120: // If counter is equal to the max # of test channels, reset it; else, proceed around again 
IF (uiLoopRcvIndex = gc.uiMaxNrDMXTestCh) THEN
	iCompareSeq[ENUM_SeqSM.Once]			:= 130;
ELSE
	uiLoopRcvIndex							:= uiLoopRcvIndex +1;
	//Next iteration
	tonTestIterGap.IN						:= TRUE;
	iCompareSeq[ENUM_SeqSM.Once]			:= 10;
 (*iCounter <> gc.usiMaxNrOfChannels*)
END_IF

130:
xDMXSeqTestInProgressOnce					:= FALSE;
iCompareSeq[ENUM_SeqSM.Once]				:= 140;

140:
IF rt_ResetTestSeq.Q AND NOT rt_RunSeqTestOnce.Q THEN
	FOR uiCounter2 := 0 TO gc.uiMaxNrDMXTestCh BY 1 DO 
		arr_diTestPNPSeqOnceLine[uiCounter2]		:= 0;
		arr_diTestNPNSeqOnceLine[uiCounter2]		:= 0;
//		arrdiTestPNPSeqOnceComplete[uiCounter2]		:= 0;
//		arrdiTestNPNSeqOnceComplete[uiCounter2]		:= 0;
		arrdiTestNPNSeqOnceCompleteProblemIndex[uiCounter2]	:= 0;
	END_FOR
	diCompTestResult							:= 0;
	iCompareSeq[ENUM_SeqSM.Once]				:= 0; (* reset to beginning *)
END_IF

END_CASE
END_ACTION

ACTION SeqTestOnceDC:
//Run Once - DMX Channels only for now

rt_RunSeqTestOnceDC();
rt_ResetTestSeqDC();

CASE iCompareSeq[ENUM_SeqSM.OnceDC] OF
	
0: // If test is triggered by user
//Trigger should be something like 
IF rt_RunSeqTestOnceDC.Q THEN
	xDMXSeqTestInProgressOnceDC				:= TRUE;
	uiLoopRcvIndex							:= cuiMinDUTIndex; 
	iCompareSeq[ENUM_SeqSM.OnceDC]			:= 10;
END_IF

10: // Zero out all comparison buffers before each comparison
IF (uiLoopRcvIndex=0) THEN
	IF xDMXSeqTestInProgressOnceDC THEN
//by default, Counter = 0 at the first initialization; it is reset at the end of this State Machine
//Clear Storage Buffers pre-test to ensure no old data interferes with current test
		FOR uiCounter4 := 0 TO gc.uiMaxNrDMXTestCh BY 1 DO
			arrxExpctdTmpPNPSeqDC[uiCounter4]		:= 0;		//should be all 0s ; PNP<>DMX
			arrxExpctdTmpNPNSeqDC[uiCounter4]		:= 0;
//			arrxExpctdTmpPNPSeqDC[uiCounter4]		:= 0;		
//			arrxExpctdTmpNPNSeqDC[uiCounter4]		:= 0;
			arrxRcvdBufferPNPSeq[uiCounter4]		:= 0;		//should be all 0s too ; PNP<>DMX	
			arrxRcvdBufferNPNSeq[uiCounter4]		:= 0;			
			g_ast.DMX[uiCounter4].IQ.xCmdOff		:= TRUE;	
		END_FOR
	iCompareSeq[ENUM_SeqSM.OnceDC]					:= 20;
	END_IF
ELSIF (uiLoopRcvIndex>0) THEN // to avoid 
	IF xDMXSeqTestInProgressOnceDC AND tonTestIterGap.Q THEN
		tonTestIterGap.IN	:= FALSE;
		//by default, Counter = 0 at the first initialization; it is reset at the end of this State Machine
		//Clear Storage Buffers pre-test to ensure no old data interferes with current test
		FOR uiCounter4 := 0 TO gc.uiMaxNrDMXTestCh BY 1 DO
			arrxExpctdTmpPNPSeqDC[uiCounter4]		:= 0;		//should be all 0s - PNP<>DMX
			arrxExpctdTmpNPNSeqDC[uiCounter4]		:= 0;
			arrxRcvdBufferPNPSeq[uiCounter4]		:= 0;		
			arrxRcvdBufferNPNSeq[uiCounter4]		:= 0;		
		END_FOR
		
	iCompareSeq[ENUM_SeqSM.OnceDC]					:= 25; // don't write the hardware value (skip 20)
	END_IF	
END_IF
	
20:	
//write 'hardware-clear' state 
g_ast.DMXHWOut									:= g_ast.DMXPhysOut;

iCompareSeq[ENUM_SeqSM.OnceDC]					:= 25;

25:
//Copy static test indices from Expected_Static - as these should still be used for comparisons
//FOR uiCounter4 := 0 TO gc.uiMaxNrDMXTestCh BY 1 DO
//	IF (arrui24VTestIndices[uiCounter4] <> 0) THEN	
		MEMCPY(srcAddr:=ADR(arrxExpctdTmpPNP24V[cuiMinDUTIndex]),destAddr:=ADR(arrxExpctdTmpPNPSeqDC[cuiMinDUTIndex]),n:=gc.uiChannelsUT);
//		MEMCPY(srcAddr:=ADR(arrxExpctdTmpNPN24V[cuiMinDUTIndex]),destAddr:=ADR(arrxExpctdTmpNPNSeqDMX[cuiMinDUTIndex]),n:=gc.uiChannelsUT);
//		MEMCPY(srcAddr:=ADR(arrxExpctdTmpPNP24V[arrui24VTestIndices[uiCounter4]]),destAddr:=ADR(arrxExpctdTmpPNPSeqDC[arrui24VTestIndices[uiCounter4]]),n:=1);
//		MEMCPY(srcAddr:=ADR(arrxExpctdTmpNPN24V[arrui24VTestIndices[uiCounter4]]),destAddr:=ADR(arrxExpctdTmpNPNSeqDC[arrui24VTestIndices[uiCounter4]]),n:=1);
//	END_IF
	
//	IF (arruiGNDTestIndices[uiCounter4] <> 0) THEN	
//		MEMCPY(srcAddr:=ADR(arrxExpctdTmpPNPGND[cuiMinDUTIndex]),destAddr:=ADR(arrxExpctdTmpPNPSeqDMX[cuiMinDUTIndex]),n:=gc.uiChannelsUT);
		MEMCPY(srcAddr:=ADR(arrxExpctdTmpNPNGND[cuiMinDUTIndex]),destAddr:=ADR(arrxExpctdTmpNPNSeqDC[cuiMinDUTIndex]),n:=gc.uiChannelsUT);
//		MEMCPY(srcAddr:=ADR(arrxExpctdTmpPNPGND[arruiGNDTestIndices[uiCounter4]]),destAddr:=ADR([arrxExpctdTmpPNPSeqDC[uiCounter4]]),n:=1);
//		MEMCPY(srcAddr:=ADR(arrxExpctdTmpNPNGND[arruiGNDTestIndices[uiCounter4]]),destAddr:=ADR(arrxExpctdTmpNPNSeqDC[arruiGNDTestIndices[uiCounter4]]),n:=1);
//	END_IF
//END_FOR

// Be careful not to overstamp existing arrays!  Right now MEMCPY is only addressing PNP24V & NPNGND

iCompareSeq[ENUM_SeqSM.OnceDC]					:= 30;

30: //Set the Expected Mask & write data to controller
//Write the first index from the specified array of indices
IF (arruiSeqTestIndicesDC[uiLoopRcvIndex] <> 0) THEN
//Also copy this specific channel index value to the comparison array
	
//Don't copy NPN indices for DC; this doesn't generally make sense
	MEMCPY(srcAddr:=ADR(arrxExpctdTmpPNP[arruiSeqTestIndicesDC[uiLoopRcvIndex]]),destAddr:=ADR(arrxExpctdTmpPNPSeqDC[arruiSeqTestIndicesDC[uiLoopRcvIndex]]),n:=SIZEOF(arrxExpctdTmpPNP[arruiSeqTestIndicesDC[uiLoopRcvIndex]]));
//	MEMCPY(srcAddr:=ADR(arrxExpctdTmpNPN[arruiSeqTestIndicesDMX[uiLoopRcvIndex]]),destAddr:=ADR(arrxExpctdTmpNPNSeqDMX[arruiSeqTestIndicesDMX[uiLoopRcvIndex]]),n:=SIZEOF(arrxExpctdTmpNPN[arruiSeqTestIndicesDMX[uiLoopRcvIndex]]));	
	
	//And Cmd - turn on - that respective channel
	g_ast.DMX[arruiSeqTestIndicesDC[uiLoopRcvIndex]].IQ.xCmdOn			:= TRUE;
	FOR uiCounter3 := cuiMinDUTIndex TO gc.uiMaxNrDMXTestCh BY 1 DO
		IF uiCounter3 <> arruiSeqTestIndicesDC[uiLoopRcvIndex] THEN
			g_ast.DMX[uiCounter3].IQ.xCmdOff	:= TRUE;	
		END_IF
	END_FOR
ELSIF (arruiSeqTestIndicesDC[uiLoopRcvIndex] = 0) THEN
	FOR uiCounter3 := cuiMinDUTIndex TO gc.uiMaxNrDMXTestCh BY 1 DO
		IF uiCounter3 <> arruiSeqTestIndicesDC[uiLoopRcvIndex] THEN
			g_ast.DMX[uiCounter3].IQ.xCmdOff	:= TRUE;	
		END_IF
	END_FOR
END_IF

iCompareSeq[ENUM_SeqSM.OnceDC]		:= 35;

35:
//Write to hardware
g_ast.DMXHWOut						:= g_ast.DMXPhysOut;

iCompareSeq[ENUM_SeqSM.OnceDC]		:= 40;

40:
//Write DMX channels
tonWriteCopyWait.IN					:= TRUE;
iCompareSeq[ENUM_SeqSM.OnceDC]		:= 50;

50:
IF tonWriteCopyWait.Q THEN
	tonWriteCopyWait.IN				:= FALSE;
	iCompareSeq[ENUM_SeqSM.OnceDC]	:= 60;
END_IF

60:
//IF there is an index for a 'Light' element, then copy that element's value to a new pair of arrays, for 'Received'
//IF arruiSeqTestIndicesDMX[uiLoopRcvIndex] <> 0 THEN
(*
FOR uiCounter6 := 0 TO gc.uiMaxNrDMXTestCh BY 1 DO 
	arr_udiMEMCPYPNPSeqOnceRcvdTmp[uiCounter6]	:= MEMCPY(srcAddr:=ADR(arrxTestChInputPNPAlias[uiCounter6]),destAddr:=ADR(arrxRcvdBufferPNPSeq[uiCounter6]),n:=SIZEOF(arrxTestChInputPNP[uiCounter6])); //bytes
	arr_udiMEMCPYNPNSeqOnceRcvdTmp[uiCounter6]	:= MEMCPY(srcAddr:=ADR(arrxTestChInputNPNAlias[uiCounter6]),destAddr:=ADR(arrxRcvdBufferNPNSeq[uiCounter6]),n:=SIZEOF(arrxTestChInputNPN[uiCounter6])); //bytes)
	//	MEMCPY(srcAddr:=ADR(arrxExpctdTmpPNP[arruiSeqTestIndices[uiLoopRcvIndex]]),destAddr:=ADR(arrxExpctdTmpPNPSeq[arruiSeqTestIndices[uiLoopRcvIndex]]),n:=1); //bytes
	//	MEMCPY(srcAddr:=ADR(arrxExpctdTmpNPN[arruiSeqTestIndices[uiLoopRcvIndex]]),destAddr:=ADR(arrxExpctdTmpNPNSeq[arruiSeqTestIndices[uiLoopRcvIndex]]),n:=1); //bytes
END_FOR
*)
//Stash
//arr_udiMEMCPYPNPSeqOnceRcvd	:= arr_udiMEMCPYPNPSeqOnceRcvdTmp;
//arr_udiMEMCPYNPNSeqOnceRcvd	:= arr_udiMEMCPYNPNSeqOnceRcvdTmp;

//END_IF

//We should also 'expect' the static indices - and if we passed the static test already - they will still be on, so grab and add those to the 'Expected' Buffer
//This is a gate to leave this state; the MEMCPY operation had to return for all values
	
(*
70:
tonReadWait.IN							:= TRUE;
iCompareSeq[ENUM_SeqSM.OnceDC]			:= 80;

80: // if wait completed, set the bit for conversion high
//Conversion Function call
IF tonReadWait.Q THEN
	tonReadWait.IN					:= FALSE;
	iCompareSeq[ENUM_SeqSM.OnceDC]	:= 90;
END_IF
*)

90:
//Run Comparos
IF iCompareStaticSM <> 90 THEN //because it uses the same iterator in StaticSM - shouldn't be the case, but this is a safeguard
	FOR uiCounter6	:= 0 TO gc.uiMaxNrDMXTestCh BY 1 DO
		arr_diTestPNPSeqOnceLineTmp[uiCounter6]			:= MEMCMP(pBuf1:=ADR(arrxExpctdTmpPNPSeqDC[uiCounter6]),pBuf2:=ADR(arrxRcvdBufferPNPSeq[uiCounter6]),n:=SIZEOF(arrxExpctdTmpPNPSeqDC[uiCounter6]));
//		arr_diTestNPNSeqOnceLineTmp[uiCounter6]			:= MEMCMP(pBuf1:=ADR(arrxExpctdTmpNPNSeqDMX[uiCounter6]),pBuf2:=ADR(arrxRcvdBufferNPNSeq[uiCounter6]),n:=SIZEOF(arrxExpctdTmpNPNSeqDMX[uiCounter6])); 
		arrdiTestPNPSeqOnceCompleteTmp[uiCounter6]		:= MEMCMP(pBuf1:=ADR(arrxExpctdTmpPNPSeqDC[cuiMinDUTIndex]),pBuf2:=ADR(arrxRcvdBufferPNPSeq[cuiMinDUTIndex]),n:=gc.uiChannelsUT); //UINTs are 16-bit/2 bytes
//		arrdiTestNPNSeqOnceCompleteTmp[uiCounter6]		:= MEMCMP(pBuf1:=ADR(arrxExpctdTmpNPNSeqDMX[cuiMinDUTIndex]),pBuf2:=ADR(arrxRcvdBufferNPNSeq[cuiMinDUTIndex]),n:=gc.uiChannelsUT); //UINTs are 16-bit/2 bytes
	END_FOR
arr_diTestPNPSeqOnceLine	:= arr_diTestPNPSeqOnceLineTmp;
arrdiTestPNPSeqOnceComplete	:= arrdiTestPNPSeqOnceCompleteTmp;
	
END_IF

(* log the error index 
IF arr_diTestPNPSeqOnce[uiLoopRcvIndex] <> 0 THEN
	memcpy(srcAddr:=uiLoopRcvIndex,destAddr:=, n:=2)
END_IF
*)

iCompareSeq[ENUM_SeqSM.OnceDC]				:= 100;

100: // If counter is equal to the max # of test channels, reset it; turn off the DMX channels that were turned on in the course of the test

IF (uiLoopRcvIndex = gc.uiMaxNrDMXTestCh) THEN
	iCompareSeq[ENUM_SeqSM.OnceDC]			:= 110;
ELSE
	uiLoopRcvIndex							:= uiLoopRcvIndex +1;
	//Next iteration
	tonTestIterGap.IN						:= TRUE;
	iCompareSeq[ENUM_SeqSM.OnceDC]			:= 10;
 (*iCounter <> gc.usiMaxNrOfChannels*)
END_IF

110:
xDMXSeqTestInProgressOnceDC					:= FALSE;
iCompareSeq[ENUM_SeqSM.OnceDC]				:= 120;

120:
IF rt_ResetTestSeqDC.Q AND NOT rt_RunSeqTestOnceDC.Q THEN
	FOR uiCounter2 := 0 TO gc.uiMaxNrDMXTestCh BY 1 DO 
		arr_diTestPNPSeqOnceLine[uiCounter2]		:= 0;
		arr_diTestNPNSeqOnceLine[uiCounter2]		:= 0;
		arrdiTestPNPSeqOnceComplete[uiCounter2]		:= 0;
		arrdiTestNPNSeqOnceComplete[uiCounter2]		:= 0;
	END_FOR
	diCompTestResult							:= 0;
	iCompareSeq[ENUM_SeqSM.OnceDC]				:= 0; (* reset to beginning *)
END_IF

END_CASE
END_ACTION

END_PROGRAM

// ---- POUs/FunctionBlocks/HelperPRG/InterfaceLink.TcPOU
PROGRAM InterfaceLink
VAR
	iResult					: INT;
	iLoopFBAnalogIn			: INT;
	iLoopFBSensor			: INT;
	iLoopFBValveSensor		: INT;
	iLoopFBDigCtrl			: INT;
	iLoopFBValveCtrl		: INT;
	uiLoopDMXCtrlI			: UINT;
	uiLoopDMXCtrlII			: UINT;
	uiLoopDebouncePNPI		: UINT;
	uiLoopDebounceNPNI		: UINT;
END_VAR

//Call all the I/O Function Blocks continuously; link to array-structs with every call;
(*
FOR iLoopFBAnalogIn := 0 TO gc.usiMaxNrOfAnalogIn BY 1 DO
	gFB.arrFB_AnalogInput[iLoopFBAnalogIn](I:=gast_AnalogInput[iLoopFBAnalogIn].I, IQ:=gast_AnalogInput[iLoopFBAnalogIn].IQ, Q=>gast_AnalogInput[iLoopFBAnalogIn].Q);
END_FOR

FOR iLoopFBSensor := 0 TO gc.usiMaxNrOfSensor BY 1 DO
	gFB.arrFB_Sensor[iLoopFBSensor](I:=gast_SensorInput[iLoopFBSensor].I, IQ:=gast_SensorInput[iLoopFBSensor].IQ, Q=>gast_SensorInput[iLoopFBSensor].Q);
END_FOR

FOR iLoopFBValveSensor := 0 TO (2*gc.usiMaxNrOfValveCtrl) BY 1 DO
	gFB.arrFB_Sensor[iLoopFBValveSensor](I:=gast_ValveSensorInput[iLoopFBValveSensor].I, IQ:=gast_ValveSensorInput[iLoopFBValveSensor].IQ, Q=>gast_ValveSensorInput[iLoopFBValveSensor].Q);
END_FOR

FOR iLoopFBDigCtrl := 0 TO gc.usiMaxNrOfSensor BY 1 DO
	gFB.arrFB_DigCtrl[iLoopFBDigCtrl](I:=gast_DigCtrlOutput[iLoopFBDigCtrl].I, IQ:=gast_DigCtrlOutput[iLoopFBDigCtrl].IQ, Q=>gast_DigCtrlOutput[iLoopFBDigCtrl].Q);
END_FOR

FOR iLoopFBValveCtrl := 0 TO gc.usiMaxNrOfValveCtrl BY 1 DO
	gFB.arrFB_ValveCtrl[iLoopFBValveCtrl](I:=gast_ValveCtrlOutput[iLoopFBValveCtrl].I, IQ:=gast_ValveCtrlOutput[iLoopFBValveCtrl].IQ, Q=>gast_ValveCtrlOutput[iLoopFBValveCtrl].Q);
END_FOR
*)
FOR uiLoopDMXCtrlI := 0 TO gc.uiMaxNrOfDMXChannel BY 1 DO
	gFB.arrFB_DMX[uiLoopDMXCtrlI](I:=g_ast.DMX[uiLoopDMXCtrlI].I, IQ:=g_ast.DMX[uiLoopDMXCtrlI].IQ, Q=>g_ast.DMX[uiLoopDMXCtrlI].Q);
END_FOR

//Expose an array of bytes that can be ultimately 'multi-linked' to hardware
FOR uiLoopDMXCtrlII := 0 TO gc.uiMaxNrOfDMXChannel BY 1 DO
	g_ast.DMXPhysOut[uiLoopDMXCtrlII]	:= g_ast.DMX[uiLoopDMXCtrlII].Q.byStatValue;
END_FOR

//Debounce PNP
FOR uiLoopDebouncePNPI	:= 0 TO gc.uiMaxNrDMXTestCh BY 1 DO
	gFB.arrFB_DebouncePNP[uiLoopDebouncePNPI](I:=g_ast.arrFBIntPNP[uiLoopDebouncePNPI].I, IQ:=g_ast.arrFBIntPNP[uiLoopDebouncePNPI].IQ, Q=>g_ast.arrFBIntPNP[uiLoopDebouncePNPI].Q);
END_FOR

//Debounce NPN
FOR uiLoopDebounceNPNI	:= 0 TO gc.uiMaxNrDMXTestCh BY 1 DO
	gFB.arrFB_DebounceNPN[uiLoopDebounceNPNI](I:=g_ast.arrFBIntNPN[uiLoopDebounceNPNI].I, IQ:=g_ast.arrFBIntNPN[uiLoopDebounceNPNI].IQ, Q=>g_ast.arrFBIntNPN[uiLoopDebounceNPNI].Q);
END_FOR

END_PROGRAM

// ---- POUs/FunctionBlocks/HelperPRG/IOParams.TcPOU
PROGRAM IOParams
VAR
	iForLoopDMXI1			: INT;
	iForLoopDMXI2			: INT;
	iForLoopDMXI3			: INT;
	iForLoopDMXI4			: INT;
	iForLoopDMXI5			: INT;
	iForLoopDMXI6			: INT;
	iForLoopDMXI7			: INT;
	iForLoopDMXI8			: INT;
	uiForLoopDMXI10			: UINT;
	uiForLoopDMXI11			: UINT;
	uiForLoopDebouncePNP	: UINT;
	uiForLoopDebounceNPN	: UINT;
END_VAR

//Link all the user-specified params to the respective Function Blocks
//RED

(*
RGB PARAMETERS - Hence, the Groups of 4 incremented in this way;

FOR iForLoopDMXI1:= 0 TO gc.uiMaxNrOfDMXChannel BY 4 DO
	g_ast.DMX[iForLoopDMXI1].I.ENWaveform		:= ENUM_I_Waveform.EN_Sin; //"50% duty cycle"
	g_ast.DMX[iForLoopDMXI1].I.fDutyCycle		:= 50; // %
	g_ast.DMX[iForLoopDMXI1].I.fLevel			:= iSlider5; //%
	g_ast.DMX[iForLoopDMXI1].I.fOffset			:= 0; // %
	g_ast.DMX[iForLoopDMXI1].I.usiBitDepth		:= 8; // 0-8, or 0-16, depending
	g_ast.DMX[iForLoopDMXI1].I.fPhase			:= 0; // %
	g_ast.DMX[iForLoopDMXI1].I.fDelay			:= 0; // %
	g_ast.DMX[iForLoopDMXI1].I.usiDelayDiv		:= 0; // which step to have delay applied
END_FOR

//GREEN
FOR iForLoopDMXI2:= 1 TO gc.uiMaxNrOfDMXChannel BY 4 DO
	g_ast.DMX[iForLoopDMXI2].I.ENWaveform		:= ENUM_I_Waveform.EN_Sin; //"50% duty cycle"
	g_ast.DMX[iForLoopDMXI2].I.fDutyCycle		:= 50; // %
	g_ast.DMX[iForLoopDMXI2].I.fLevel			:= iSlider6; //%
	g_ast.DMX[iForLoopDMXI2].I.fOffset			:= 0; // %
	g_ast.DMX[iForLoopDMXI2].I.usiBitDepth		:= 8; // 0-8, or 0-16, depending
	g_ast.DMX[iForLoopDMXI2].I.fPhase			:= 0; // %
	g_ast.DMX[iForLoopDMXI2].I.fDelay			:= 0; // %
	g_ast.DMX[iForLoopDMXI2].I.usiDelayDiv		:= 0; // which step to have delay applied
END_FOR

//BLUE
FOR iForLoopDMXI3:= 2 TO gc.uiMaxNrOfDMXChannel BY 4 DO
	g_ast.DMX[iForLoopDMXI3].I.ENWaveform		:= ENUM_I_Waveform.EN_Sin; //"50% duty cycle"
	g_ast.DMX[iForLoopDMXI3].I.fDutyCycle		:= 50; // %
	g_ast.DMX[iForLoopDMXI3].I.fLevel			:= iSlider7; //%
	g_ast.DMX[iForLoopDMXI3].I.fOffset			:= 0; // %
	g_ast.DMX[iForLoopDMXI3].I.usiBitDepth		:= 8; // 0-8, or 0-16, depending
	g_ast.DMX[iForLoopDMXI3].I.fPhase			:= 0; // %
	g_ast.DMX[iForLoopDMXI3].I.fDelay			:= 0; // %
	g_ast.DMX[iForLoopDMXI3].I.usiDelayDiv		:= 0; // which step to have delay applied
END_FOR

//WHITE
FOR iForLoopDMXI4:= 3 TO gc.uiMaxNrOfDMXChannel BY 4 DO
	g_ast.DMX[iForLoopDMXI4].I.ENWaveform		:= ENUM_I_Waveform.EN_Sin; //"50% duty cycle"
	g_ast.DMX[iForLoopDMXI4].I.fDutyCycle		:= 50; // %
	g_ast.DMX[iForLoopDMXI4].I.fLevel			:= iSlider8; //%
	g_ast.DMX[iForLoopDMXI4].I.fOffset			:= 0; // %
	g_ast.DMX[iForLoopDMXI4].I.usiBitDepth		:= 8; // 0-8, or 0-16, depending
	g_ast.DMX[iForLoopDMXI4].I.fPhase			:= 0; // %
	g_ast.DMX[iForLoopDMXI4].I.fDelay			:= 0; // %
	g_ast.DMX[iForLoopDMXI4].I.usiDelayDiv		:= 0; // which step to have delay applied
END_FOR


FOR iForLoopDMXI5	:= 0 TO gc.uiMaxNrOfDMXChannel BY 4 DO 
	g_ast.DMX[iForLoopDMXI5].I.fFrequency		:= iSlider1; //Hz
END_FOR

FOR iForLoopDMXI6	:= 0 TO gc.uiMaxNrOfDMXChannel BY 4 DO 
	g_ast.DMX[iForLoopDMXI6].I.fFrequency		:= iSlider2; //Hz
END_FOR

FOR iForLoopDMXI7	:= 0 TO gc.uiMaxNrOfDMXChannel BY 4 DO 
	g_ast.DMX[iForLoopDMXI7].I.fFrequency		:= iSlider3; //Hz
END_FOR

FOR iForLoopDMXI8	:= 0 TO gc.uiMaxNrOfDMXChannel BY 4 DO 
	g_ast.DMX[iForLoopDMXI8].I.fFrequency		:= iSlider4; //Hz
END_FOR
*)

FOR uiForLoopDMXI10:= 0 TO gc.uiDUTConfigCountSplit BY 1 DO
	g_ast.DMX[uiForLoopDMXI10].I.fFrequency		:= 0;
	g_ast.DMX[uiForLoopDMXI10].I.ENWaveform		:= ENUM_I_Waveform.EN_GateCtrl;
	g_ast.DMX[uiForLoopDMXI10].I.ENValRange		:= ENUM_I_ValRange.EN_8Bit;
	g_ast.DMX[uiForLoopDMXI10].I.fDutyCycle		:= 100; // %
	g_ast.DMX[uiForLoopDMXI10].I.fLevel			:= 100; //%
	g_ast.DMX[uiForLoopDMXI10].I.fOffset		:= 0; // %
	g_ast.DMX[uiForLoopDMXI10].I.usiBitDepth	:= 8; // 0-8, or 0-16, depending
	g_ast.DMX[uiForLoopDMXI10].I.fPhase			:= 0; // %
	g_ast.DMX[uiForLoopDMXI10].I.fDelay			:= 0; // %
	g_ast.DMX[uiForLoopDMXI10].I.usiDelayDiv	:= 0; // which step to have delay applied
//Channels for Configuration of testing on other DMX Channels;
END_FOR

FOR uiForLoopDMXI10:= gc.uiChannelSplitCount TO gc.uiMaxNrOfDMXChannel BY 1 DO
	g_ast.DMX[uiForLoopDMXI10].I.fFrequency		:= 0;
	g_ast.DMX[uiForLoopDMXI10].I.ENWaveform		:= ENUM_I_Waveform.EN_GateConfig;
	g_ast.DMX[uiForLoopDMXI10].I.ENValRange		:= ENUM_I_ValRange.EN_8Bit;
	g_ast.DMX[uiForLoopDMXI10].I.fDutyCycle		:= 100; // %
	g_ast.DMX[uiForLoopDMXI10].I.fLevel			:= 100; //%
	g_ast.DMX[uiForLoopDMXI10].I.fOffset		:= 0; // %
	g_ast.DMX[uiForLoopDMXI10].I.usiBitDepth	:= 8; // 0-8, or 0-16, depending
	g_ast.DMX[uiForLoopDMXI10].I.fPhase			:= 0; // %
	g_ast.DMX[uiForLoopDMXI10].I.fDelay			:= 0; // %
	g_ast.DMX[uiForLoopDMXI10].I.usiDelayDiv	:= 0; // which step to have delay applied
//Channels for Configuration of testing on other DMX Channels;
END_FOR

//Input Debounce Params PNP
FOR uiForLoopDebouncePNP	:= 0 TO gc.uiMaxNrDMXTestCh BY 1 DO
	g_ast.arrFBIntPNP[uiForLoopDebouncePNP].I.tOnDelay	:= T#0S;
	g_ast.arrFBIntPNP[uiForLoopDebouncePNP].I.tOffDelay	:= T#10MS;
END_FOR

//Input Debounce Params NPN
FOR uiForLoopDebounceNPN	:= 0 TO gc.uiMaxNrDMXTestCh BY 1 DO
	g_ast.arrFBIntNPN[uiForLoopDebounceNPN].I.tOnDelay	:= T#0S;
	g_ast.arrFBIntNPN[uiForLoopDebounceNPN].I.tOffDelay	:= T#3MS;
END_FOR

//Read the CSV Parameters into the DMX FBs - via the "mediating" Config arrays
FOR uiForLoopDMXI11:= 0 TO gc.uiMaxNrOfDMXChannel BY 1 DO
	g_ast.DMX[DMXTest.arr_uiRecipeIndex[uiForLoopDMXI11]].I.usiInputConfig	:= 	DMXTest.arr_usiRecipeSetting[uiForLoopDMXI11];
END_FOR

END_PROGRAM

// ---- POUs/FunctionBlocks/FB_DMX.TcPOU
FUNCTION_BLOCK FB_DMX
VAR_INPUT
	I	: typDMXInput;
END_VAR

VAR_IN_OUT
	IQ	: typDMXInOut;
END_VAR

VAR_OUTPUT
	Q	: typDMXOutput;
END_VAR

VAR
//	uiOpStatus			: UINT;
	iWaveSelectSM		: INT;
	uiTimeCycleSM		: UINT;
	uiDelayShiftSM		: UINT;
	uiTimeShiftSM		: UINT;
	uiDeviceSM			: UINT;
	uiModeCtrlSM		: UINT;

	uiPulseCount		: UINT;
	fPhaseShift			: REAL;
	fDelayShift			: REAL;
	tTimeShift			: TIME;
	tPhaseShift			: TIME;
	tDelayShift			: TIME;

	fLevelShift			: REAL;
	fOffsetShift		: REAL;	
	tOnPulse			: TON;
	tOnShift			: TON;
	
	tonFnWindow			: TON;
	tonSqDutyCyc		: TON;
	fDutyCycle			: REAL;
	
	fFnGenerValTempSin	: LREAL;
	fFnGenerValAdj		: REAL; //Adjusted channel value: rounded, clamped, scaled per the input parameters for the channel
	
	rt_FnRisEdge		: R_TRIG;
	
	cfLoFnVal			: REAL	:= 0; // min function value from function generator
	cfHiFnVal			: REAL	:= 2; // max function value from function generator
	
	fFnWindowET			: REAL;
	tPeriod				: TIME;
	tonRunning			: TON;
	tonRunningSH		: TON;
	iClockSM			: INT;
	iFnSampleHoldSM		: INT;
	
	//not currently used:	
	tonFnSomethingElse	: TON;
	
	fPeriod				: REAL;
	tFnWindowET			: TIME;
END_VAR

//Compute Regular Trigger/Pulse train:
CASE uiTimeCycleSM OF
	
0: //Execute timer
tOnPulse.IN		:= TRUE;
uiTimeCycleSM	:= 10;

10:  //Wait for timer completion ; reset timer
IF tOnPulse.Q THEN
	tOnPulse.IN		:= FALSE;
	uiTimeCycleSM	:= 0;
END_IF

END_CASE

//calculate time shift
tPhaseShift	:= REAL_TO_TIME(fPhaseShift);

tDelayShift	:= REAL_TO_TIME(fDelayShift);

tTimeShift	:= tPhaseShift + tDelayShift;

//Phase Shift Function
fPhaseShift	:= (I.fPhase/100)(*percentage*)*fPeriod;

//Delay Shift also uses this SM (State Machine) in order to apply fDelayShift on the appropriate step
CASE uiDelayShiftSM OF
	
0:
IF tOnPulse.Q THEN
	uiPulseCount	:= uiPulseCount + 1;
	uiDelayShiftSM	:= 10;
END_IF

10: // State to apply the Delay Time Shift

//Reset the Pulse Counter if it is equivalent to the delay divisor ; and shift state to apply the delay on that "step"
IF uiPulseCount = I.usiDelayDiv THEN
	uiPulseCount	:= 0;
	//Delay Shift Function
	IF I.fFrequency <> 0 THEN
		fDelayShift	:= (I.fDelay/100)(*percentage*)*fPeriod;
	END_IF
ELSIF (I.usiDelayDiv = 0) THEN
	uiPulseCount	:= 0;
ELSE (* uiPulseCount <> I.usiDelayDiv THEN *)  
	fDelayShift		:= 0; (* Delay Shift always = 0 when it is on a step that is not equal to I.usiDelayDiv *)
	uiDelayShiftSM	:= 0; (* return to increment pulse counter *)
END_IF

END_CASE

//This SM sees rising edge from pulse; applies time shift (even if time shift = 0)
CASE uiTimeShiftSM OF 
	
0: // If there is a rising edge from the Pulse clock, implement tonShift, a delay
IF tOnPulse.IN THEN
	tOnShift.IN	:= TRUE;
	uiTimeShiftSM	:= 10;
END_IF

10:
IF tOnShift.Q THEN
	tOnShift.IN		:= FALSE;
	uiTimeShiftSM	:= 0;
END_IF

END_CASE


//level shift code:
//offset adjusts 'bottom' rail, level adjusts 'top' rail;
//bit depth specifies the 'fine-ness' of the value range for the output
//Sets the IQ - basically modifies the user input 'I'

IF I.ENValRange = ENUM_I_ValRange.EN_8Bit THEN //accept the user input params
	IQ.uiMaxChannelVal	:= 255;
ELSIF I.ENValRange = ENUM_I_ValRange.EN_16Bit THEN //accept the user input params
	IQ.uiMaxChannelVal	:= 65535;
END_IF

//perhaps have a 'preset' condition like this, for Boolean:
//Sets the IQ - basically modifies the user input 'I'
IF (I.ENWaveform = ENUM_I_Waveform.EN_GateCtrl) OR (I.ENWaveform = ENUM_I_Waveform.EN_GateConfig) OR (I.usiBitDepth = 1) THEN
	IQ.fLevel		:= Map(fArg:=100(*%*),fInMin:=0,fInMax:=100,fOutMin:=IQ.uiMinChannelVal,fOutMax:=IQ.uiMaxChannelVal);
	IQ.usiBitDepth	:= 1;
	IQ.fOffset		:= Map(fArg:=0(*%*),fInMin:=0,fInMax:=100,fOutMin:=IQ.uiMinChannelVal,fOutMax:=IQ.uiMaxChannelVal);
ELSE (* not Boolean/Gate operation *)
	IQ.fLevel		:= Map(I.fLevel,0,100,0,IQ.uiMaxChannelVal); // scale % to 255
	IQ.usiBitDepth	:= I.usiBitDepth; 
	IQ.fOffset		:= Map(I.fOffset,0,100,0,IQ.uiMaxChannelVal); // scale % to 255
END_IF

//Return a mapped value, clamped to a 'nearest value' governed by the bit depth
//Check IQ.fFnGenerValRtn range; if it's from the sin function, use input range [0,2]; else use [0,100]

Q.byStatValue		:= REAL_TO_BYTE(Q.fFnGeneratorVal);
IQ.byMinChanVal		:= UINT_TO_BYTE(IQ.uiMinChannelVal);
IQ.byMaxChanVal		:= UINT_TO_BYTE(IQ.uiMaxChannelVal);

tFnWindowET			:= tonRunning.ET;
fFnWindowET			:= TIME_TO_REAL(tFnWindowET);

CASE iWaveSelectSM OF

// Wave Select State Machine needs to output a "function" value.  This can be continuously generated.  In all cases, let's say for example's sake we are using something like "f(x) = sin(x)".  
// The values of the function output should be scaled from (0,2) of (-1,1).  The scaled value should be input to the function below that maps and re-scales this function output, 
// to fit the range of user parameters (level, offset, bit depth) specified.  Perhaps this for all function outputs - 

0: // Default to zero state for this SM, then go to the relevant function generator (enumerator) state
IF rt_FnRisEdge.Q THEN
	tonFnWindow.IN	:= TRUE;
	iWaveSelectSM	:= I.ENWaveform;
END_IF

ENUM_I_Waveform.EN_Square:
IF I.fFrequency = 0 THEN
	IQ.fFnGenerValRtn	:= IQ.fLevel; // Set it to the permissible max of the range
ELSE (* I.fFrequency <> 0 *)
	tonSqDutyCyc.IN		:= TRUE;
	IQ.fFnGenerValRtn	:= 255*BOOL_TO_LREAL(tonSqDutyCyc.IN);
	iWaveSelectSM		:= 15;
END_IF

15:
IF tonSqDutyCyc.Q THEN
	tonSqDutyCyc.IN		:= FALSE;
	iWaveSelectSM		:= ENUM_I_Waveform.EN_Square;
END_IF

//Basically the same as 'Square' but no 'duty cycle'
ENUM_I_Waveform.EN_GateConfig (* Note 8-bit Only *):

// Relay NC condition = PNP; Relay 'NO' condition = NPN
// Otherwise, DMX Function Block should function normally
IF (I.usiInputConfig <= 127) THEN
	IQ.fFnGenerValRtn		:= IQ.fOffset;
ELSIF (I.usiInputConfig > 127) THEN
	IQ.fFnGenerValRtn		:= IQ.fLevel;
END_IF

Q.fFnGeneratorVal		:= IQ.fFnGenerValRtn; // Set it to the permissible max of the range

ENUM_I_Waveform.EN_GateCtrl:
IF IQ.xCmdOn THEN
	IQ.xCmdOn			:= FALSE;
	IQ.fFnGenerValRtn	:= IQ.fLevel;
END_IF

IF IQ.xCmdOff THEN
	IQ.xCmdOff			:= FALSE;
	IQ.fFnGenerValRtn	:= IQ.fOffset;
END_IF

Q.fFnGeneratorVal		:= IQ.fFnGenerValRtn; // Set it to the permissible max of the range

ENUM_I_Waveform.EN_Sin:
IF I.ENWaveform = ENUM_I_Waveform.EN_Sin THEN
	Q.fFnGeneratorVal		:= MapClamp(IQ.fFnGenerValRtn,cfLoFnVal,cfHiFnVal,IQ.fOffset,IQ.fLevel,IQ.usiBitDepth);
ELSE
	Q.fFnGeneratorVal		:= MapClamp(IQ.fFnGenerValRtn,IQ.fOffset,IQ.fLevel,IQ.fOffset,IQ.fLevel,IQ.usiBitDepth);
END_IF

tFnWindowET			:= tonRunning.ET;
fFnWindowET			:= TIME_TO_REAL(tFnWindowET);

IQ.fFnGenerValTempSin	:= (2*gc.fPi*I.fFrequency*fFnWindowET);

//y(t)=sin(2*pi*f*t)
(*
CASE iFnSampleHoldSM OF
	
0:
tonRunningSH.IN		:= TRUE;
iFnSampleHoldSM		:= 10;

10:
IF tonRunningSH.Q THEN
	tonRunningSH.IN		:= FALSE;
	tFnWindowET			:= tonRunning.ET;
	fFnWindowET			:= TIME_TO_REAL(tFnWindowET);
	iFnSampleHoldSM	:= 0;
END_IF

END_CASE
*)

ENUM_I_Waveform.EN_Triangle:
Q.fFnGeneratorVal	:= 2; //set function value high initially, advance SM

iWaveSelectSM		:= ENUM_I_Waveform.EN_SubTriFall;

ENUM_I_Waveform.EN_SubTriFall:

//use 2 as the function value (that is the range of the function)
IF fPeriod <> 0 THEN
	Q.fFnGeneratorVal	:= Q.fFnGeneratorVal - ((2 / (fPeriod*0.5))*fFnWindowET);
END_IF

IF Q.fFnGeneratorVal = 0 THEN
	iWaveSelectSM		:= ENUM_I_Waveform.EN_SubTriRise;
END_IF

//use 2 as the function value (that is the range of the function)
ENUM_I_Waveform.EN_SubTriRise:
IF fPeriod <> 0 THEN
	Q.fFnGeneratorVal	:= Q.fFnGeneratorVal + ((2 / (fPeriod*0.5))*fFnWindowET);
END_IF

IF Q.fFnGeneratorVal = 2 THEN
	iWaveSelectSM		:= ENUM_I_Waveform.EN_Triangle;
END_IF
	
END_CASE
	
//ENUM_I_Waveform.EN_Ramp:
//function output range from (0,255) - level/offset/depth transformation (for scaling) happens separately

//ENUM_I_Waveform.EN_Rand:
//function output range from (0,255) - level/offset/depth transformation (for scaling) happens separately

//ENUM_I_Waveform.EN_Saw:
//function output range from (0,255) - level/offset/depth transformation (for scaling) happens separately

(*
CASE uiModeCtrlSM OF
	
//ENUM_I_OpMode.EN_Cycle:

ENUM_IQ_OpMode.EN_Cycle:


ENUM_IQ_OpMode.EN_LatchOn:

ENUM_IQ_OpMode.EN_OneShot:


END_CASE*)

//crufty - may be useful in future cleaning up of this FB, or not
(*
ELSIF Q.xGate (* or Function Output *) THEN
	Q.byStatValue		:= REAL_TO_BYTE(Q.fFnGeneratorVal);
ELSE (*<> Q.xGate*) (* "Offset" equivalent to the 'recipe'-adjusted 'zero' *)
	Q.byStatValue		:= REAL_TO_BYTE(IQ.fOffset);	
END_IF
*)


CASE iClockSM OF
	
0: // Start clock
tonRunning.IN	:= TRUE;
iClockSM	:= 10;

10:
IF tonRunning.Q THEN
	tonRunning.IN	:= FALSE;
	iClockSM		:= 0;
END_IF

END_CASE

IF I.fFrequency <> 0 THEN
	fPeriod		:= f_to_Period(I.fFrequency);
END_IF

tPeriod			:= REAL_TO_TIME(1000*fPeriod);

//Function Calls / Parameterization
rt_FnRisEdge(CLK	:= tOnShift.IN);
tOnPulse();
tOnPulse.PT		:= tPeriod;
tOnShift(PT	:= tTimeShift / 2);

//tonFnSomethingElse(PT	:= (REAL_TO_TIME(f_to_Period(I.fFrequency)) - tOnPulse.PT - tOnShift.PT (*- T#1MS*))); // Used for cycle mode; cycle should reset before the next 'pulse' occurs
tonFnWindow(PT	:= tPeriod); // Only dependent on period

IF I.fFrequency <> 0 THEN
	fDutyCycle	:= ((I.fDutyCycle/100) * TIME_TO_REAL(tonFnWindow.PT)); // % of the time window that the value is to be held high	
END_IF
tonSqDutyCyc();
tonSqDutyCyc.PT	:= REAL_TO_TIME(fDutyCycle);
tonRunning(PT	:= T#24H);
tonRunningSH(PT	:= T#1MS); // Preset time for how quickly to sample the ET value from 'tonRunning' - how quickly does SIN "Sample & Hold" function refresh?

END_FUNCTION_BLOCK

// ---- POUs/Functions/Map.TcPOU
FUNCTION Map : REAL
VAR_INPUT
	fArg		: REAL; //x
	fInMin		: REAL;
	fInMax		: REAL;
	fOutMin		: REAL;
	fOutMax		: REAL;	
END_VAR
VAR
END_VAR

IF (fInMax - fInMin) <> 0 THEN
	Map := (((fArg - fInMin) * (fOutMax - fOutMin)) / (fInMax - fInMin)) + fOutMin;
END_IF

END_FUNCTION

// ---- POUs/Functions/MapClamp.TcPOU
FUNCTION MapClamp : REAL
VAR_INPUT
	flArg				: LREAL; //fFnGenChanVal
	flInMin				: LREAL;
	flInMax				: LREAL;
	flOutMin			: LREAL;
	flOutMax			: LREAL;
	usiBitDepth			: USINT;
END_VAR
VAR
	flValueRange		: LREAL;
	flOutputIncrement	: LREAL;
	diOutputIncrement	: DINT;
	flUnroundedVal		: LREAL;
	diUnroundedVal		: DINT;
	flMapClampFloor		: LREAL;
	flMapClampTemp		: LREAL;
END_VAR

IF (flInMax - flInMin) <> 0 THEN
	flUnroundedVal := (((flArg - flInMin) * (flOutMax - flOutMin)) / (flInMax - flInMin)) + flOutMin;
END_IF

//Basically a sub-function (possibly could be written as a separate function that is called) to compute the nearest value for the output, based on the user input params
flValueRange	:= flOutMax - flOutMin; //Entire possible range of output values;

flOutputIncrement	:= flValueRange/EXPT(2,usiBitDepth);
diOutputIncrement	:= LREAL_TO_DINT(flOutputIncrement);

diUnroundedVal		:= LREAL_TO_INT(flUnroundedVal);

IF flOutputIncrement <> 0 THEN //avoid div by 0
	flMapClampFloor	:= FLOOR(flUnroundedVal / flOutputIncrement);//Truncate? UnroundedValue, add one increment
END_IF

IF flOutputIncrement <> 0 THEN //avoid div by 0
	IF (diUnroundedVal MOD diOutputIncrement) >= (0.5 * flOutputIncrement) THEN
		MapClamp	:=	(flMapClampFloor * flOutputIncrement) + flOutputIncrement;		//Truncate? UnroundedValue, add one increment 
	ELSIF (diUnroundedVal MOD diOutputIncrement) < (0.5 * flOutputIncrement) THEN
		MapClamp	:=	(flMapClampFloor * flOutputIncrement);
	END_IF
END_IF

IF MapClamp > flOutMax THEN
	MapClamp	:= flOutMax;
ELSIF MapClamp < flOutMin THEN
	MapClamp	:= flOutMin;	
END_IF

END_FUNCTION

// ---- POUs/Functions/f_to_Period.TcPOU
FUNCTION f_to_Period : REAL
VAR_INPUT
	fFrequency : REAL;
END_VAR
VAR	
	fFracOfTime			: REAL;
	fReferenceTimeTemp	: REAL;	
END_VAR

IF fFrequency <> 0 THEN
	fFracOfTime	:= (1/fFrequency);
END_IF

fReferenceTimeTemp	:= TIME_TO_REAL(T#1MS);

f_to_Period	:= fReferenceTimeTemp * fFracOfTime;

END_FUNCTION

// ---- POUs/Functions/SclBytePNP.TcPOU
FUNCTION SclBytePNP : BYTE
VAR_INPUT
	byUnscaled	: BYTE;
END_VAR
VAR
END_VAR

IF byUnscaled = 0 THEN
	SclBytePNP	:= 0;
ELSE
	SclBytePNP	:= 255;
END_IF

END_FUNCTION

// ---- GlobalTextList.TcGTLO
TEXTLIST GlobalTextList
  441 = '%i'
  266 = '%S'
  803 = '%s'
  91 = '(Local) Filepath of\nRecipe (.csv):\n(Tap to Edit)'
  118 = '+'
  251 = 'ack'
  1 = 'Ack!'
  454 = 'BuffCompare FALSE'
  804 = 'Channel Start'
  57 = 'Complete Filepath:'
  840 = 'Complete Filepath;'
  453 = 'Config End Channel #:%i'
  73 = 'Config End Channel #:%s'
  900 = 'Config File End Ch. #:%i'
  725 = 'Config File End Ch.#: %i'
  346 = 'Config File Start Ch #:%i'
  297 = 'Config File Start Ch.#: %i'
  67 = 'Config File Start Ch.#:%i'
  332 = 'Config Start Ch \n(HW Add.) #:%i'
  965 = 'Config Start Ch (HW Add.) #:%i'
  180 = 'Config Start Channel #:%i'
  757 = 'Config Start Channel #:%s'
  636 = 'Current\nIndex: %i'
  847 = 'Current Index: %i'
  982 = 'Data Field #1: %s'
  319 = 'DUT (HW) End Ch.#: %i'
  398 = 'DUT (HW) End Ch.#:%i'
  829 = 'DUT (HW) Start Ch.#: %i'
  560 = 'DUT End Ch.#(HW):%i'
  500 = 'DUT End Ch.#: %i'
  135 = 'DUT End Ch.#:%i'
  818 = 'DUT End Channel #:%i'
  326 = 'DUT End Channel #:%s'
  627 = 'DUT Start Ch.# (HW):%i'
  795 = 'DUT Start Ch.#: %i'
  115 = 'DUT Start Ch.#:%i'
  999 = 'DUT Start Channel #:%i'
  290 = 'DUT Start Channel #:%s'
  106 = 'End Channel #:'
  696 = 'End Channel#:'
  758 = 'Ending Index:'
  841 = 'File Date-Time:'
  926 = 'File Directory:'
  675 = 'File Extension:'
  200 = 'Filepath of Recipe (.csv):\n(Tap to Edit)'
  205 = 'Global Buffer (0=OK)'
  868 = 'Global Result'
  567 = 'Global Result: %s'
  490 = 'HW End Address Ch.#: %i'
  48 = 'HW Start Address Ch.#: %i'
  155 = 'ID# of \nUUT (Unit Under Test):'
  886 = 'ID# of UUT\n(Unit Under Test):'
  488 = 'ID# of UUT (Unit Under Test):'
  695 = 'Invert Recipe Settings'
  651 = 'Invert Recipe Settings\n(+ Set Config)'
  520 = 'Invert Recipe Settings\n+ Set Config!'
  220 = 'Invert Recipe Settings (+ Set Config)'
  156 = 'Invert Recipe Settings(+ Set Config)'
  865 = 'L Filepath:'
  96 = 'Lit = Test In Progress'
  544 = 'Load Recipe File'
  129 = 'Load Recipe File & \nSet Input Configuration'
  228 = 'Load Recipe File & +'
  399 = 'loading'
  427 = 'Local Filename of\nLast Saved Result File (.csv):'
  673 = 'Local Filename of\nResult File (.csv):'
  756 = 'Local Filename of Last\nSaved Result File (.csv):'
  742 = 'Local Filename of Last\nSaved Result File:'
  831 = 'Local Filepath of\nLoaded Recipe (.csv):'
  764 = 'Local Filepath of\nLoaded Recipe (.csv):\n(Tap to Edit)'
  553 = 'Local Filepath of\nResult File (.csv):'
  316 = 'Local Filepath of \nRecipe (.csv):'
  483 = 'Local Filepath of Loaded Recipe (.csv):'
  34 = 'Local Filepath of Recipe .csv:'
  60 = 'Local Filepath ofLoaded Recipe (.csv):'
  487 = 'Local Filepath:'
  780 = 'Read File into PLC'
  884 = 'Read File into PLC & Set Input Configuration'
  85 = 'Reset DC Test'
  587 = 'Reset DMX Test'
  472 = 'Reset Motor Test'
  191 = 'Reset Seq DMX Test'
  698 = 'Reset Test'
  592 = 'Reset Test/Clear Buffers'
  724 = 'Result File Directory:'
  28 = 'Run DC Test'
  631 = 'Run DMX Test'
  526 = 'Run Motor Test'
  903 = 'Run Multi-Channel Test'
  199 = 'Run Seq DMX Test'
  637 = 'Run Seq Test'
  291 = 'Run SeqTest'
  830 = 'Run Static Test'
  593 = 'Run Test'
  429 = 'Save Result File'
  846 = 'Save Results to File'
  663 = 'Set all DUT Values to:'
  835 = 'Set Input Configuration'
  599 = 'Set Routing per File'
  11 = 'Set Routing Relays'
  997 = 'setting config...'
  8 = 'Start Channel'
  568 = 'Start Channel #:'
  752 = 'Starting Index:'
  149 = 'Table of Channels\nw/ Discrepancies:'
  442 = 'Table of Channels w/ Issues:'
  342 = 'Table of ChannelsDiscrepancies'
  496 = 'Test End Channel #:'
  2 = 'Test End Channel #:%s'
  863 = 'Test Start Channel #:'
  213 = 'Test Start Channel #:%s'
  652 = 'Write Results to File'
END_TEXTLIST

// ---- VISUs/Visualization.TcVIS
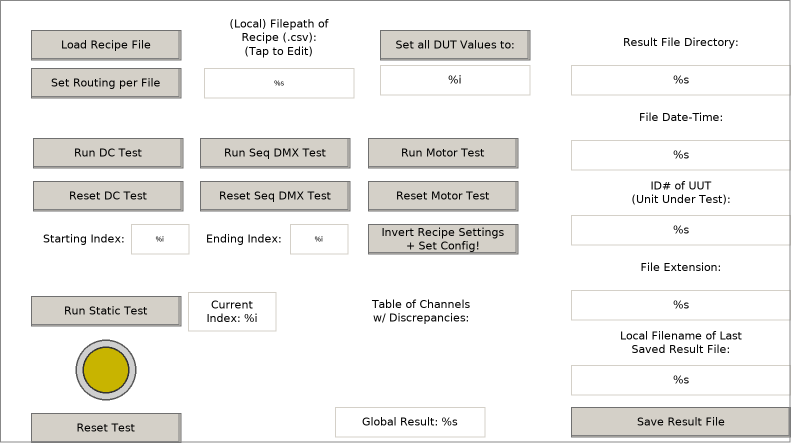
VISUALIZATION Visualization  // 791x443
    Button (31,30 150x30), "Load Recipe File", invisible if: DMXTest.iParseFile<>0
        tap P_TextModeRead.r_tFileChg.CLK
    Label (204,9 150x57), "(Local) Filepath of Recipe (.csv): (Tap to Edit)"
    Textfield (204,68 150x30), "%s", text variable: P_TextModeRead.sFilePathHMI
        OnMouseClick: write the text variable via Edit
    Textfield (335,407 150x30), "Global Result: %s"
    Label (356,296 130x30), "Table of Channels w/ Discrepancies:"
    Label (571,177 220x31), "ID# of UUT (Unit Under Test):"
    Textfield (571,215 220x30), "%s", text variable: P_TextModeWrite.sDUTIDNr
        OnMouseClick: write the text variable via VisuDialogs.Keypad
    Button (571,407 220x30), "Save Result File"
        tap P_TextModeWrite.r_tSaveResultFile.CLK
    Label (571,327 220x31), "Local Filename of Last Saved Result File:"
    Textfield (571,365 220x30), "%s", text variable: P_TextModeWrite.sFileName
    Label (571,102 220x31), "File Date-Time:"
    Textfield (571,140 220x30), "%s", text variable: P_TextModeWrite.sTimestamp
        tap P_TextModeWrite.r_tUpdateTimestamp.CLK p3779583253=TRUE
    Label (571,27 220x31), "Result File Directory:"
    Label (571,252 220x31), "File Extension:"
    Textfield (571,290 220x30), "%s", text variable: P_TextModeWrite.sFileExtension
        OnMouseClick: write the text variable via VisuDialogs.Keypad
    Textfield (571,65 220x30), "%s", text variable: P_TextModeWrite.sFileDir
        OnMouseClick: write the text variable via VisuDialogs.Keypad
    Lamp1 (71,335 70x70), variable: DMXTest.xDMXSeqTestInProgressOnce, style: Lamp-Lamp1-Yellow
    Button (31,296 150x30), "Run Static Test"
        tap DMXTest.rt_RunStaticTest.CLK
    Button (31,413 150x30), "Reset Test", invisible if: DMXTest.iCompareStaticSM<>120
        tap DMXTest.rt_ResetTest.CLK p3779583253=TRUE
    Button (31,68 150x30), "Set Routing per File", invisible if: DMXTest.iSetConfig<>0
        tap DMXTest.r_tSetConfig.CLK
    Textfield (188,292 88x39), "Current Index: %i", text variable: DMXTest.uiLoopRcvIndex
    Button (380,30 150x30), "Set all DUT Values to:"
        tap DMXTest.r_tSetDUTVal.CLK
    Textfield (380,65 150x30), "%i", text variable: DMXTest.usiDUTVal
        OnMouseClick: write the text variable via InputWithLimits, min 0, max 255
    Button (200,138 150x30), "Run Seq DMX Test"
        tap DMXTest.rt_RunSeqTestOnce.CLK p3779583253=TRUE
    Button (200,181 150x30), "Reset Seq DMX Test"
        tap DMXTest.rt_ResetTestSeq.CLK p3779583253=TRUE
    Button (33,138 150x30), "Run DC Test"
        tap DMXTest.rt_RunSeqTestOnceDC.CLK p3779583253=TRUE
    Button (33,181 150x30), "Reset DC Test"
        tap DMXTest.rt_ResetTestSeqDC.CLK p3779583253=TRUE
    Button (368,138 150x30), "Run Motor Test"
    Button (368,181 150x30), "Reset Motor Test"
    Textfield (131,224 58x30), "%i", text variable: DMXTest.uiStartingIndex
        OnMouseClick: write the text variable via Edit
    Textfield (290,224 58x30), "%i", text variable: DMXTest.uiEndingIndex
        OnMouseClick: write the text variable via Edit
    Label (44,225 80x28), "Starting Index:"
    Label (204,225 80x28), "Ending Index:"
    Button (368,224 150x30), "Invert Recipe Settings + Set Config!"
        tap DMXTest.R_TInvertRecipe.CLK p3779583253=TRUE
END_VISUALIZATION
